ABB RobotStudio station: Solution_20200508-184500.rsstn

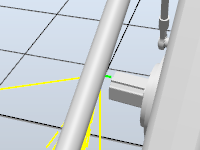
Station Solution (saved by RobotStudio 7.0.8743.626)
Controller Controller
  mechanical unit ROB_1: IRB120_3_58__01, 6 joints, base frame (-200, 0, 800) mm
  mechanical unit ROB_2: IRB120_3_58__01_2, 6 joints, base frame (200, 0, 800) mm, rotated rx 0 ry 0 rz 180 deg
  mechanical unit ROB_3: IRB760_450_318__01, 6 joints, base frame (0, 4000, 0) mm
Layout (positions relative to the parent item):
  - IRB120_3_58__01 [mechanism, from Robots\IRB120_3_58_G_01.rslib] at (-200, 0, 800) mm; joint values [0, -0.7948, 0.351, 0, 2.0145, 0] (rad or m)
  - IRB120_3_58__01_2 [mechanism, from Robots\IRB120_3_58_G_01.rslib] at (200, 0, 800) mm, rotated rx 0 ry 0 rz 180 deg; joint values [0, -0.7948, 0.351, 0, 2.0145, 0] (rad or m)
  - IRB760_450_318__01 [mechanism, from Robots\IRB760_450_318__01.rslib] at (0, 4000, 0) mm; joint values [-0.1057, 0.2404, 0.623, -1.118] (rad or m)
  - Part_1 [part]
  - Tool_1 [mechanism] at (-150, 0, 1400) mm, rotated rx 180 ry 0 rz 180 deg
      TCP Tool1 at (0, 0, 0) mm
      links: SimpleGripper
  - Tool_2 [mechanism] at (150, 0, 1400) mm, rotated rx 180 ry 0 rz 0 deg
      TCP Tool_2 at (0, 0, 0) mm
      links: SimpleGripper
  - Tool_3 [mechanism] at (1980, 3790, 1000) mm, rotated rx 180 ry 0 rz -122 deg
      TCP Tool_3 at (0, 0, 0) mm
      links: SimpleGripper
Attachment: Tool_1 is attached to IRB120_3_58__01 / Link6
Attachment: Tool_2 is attached to IRB120_3_58__01_2 / Link6
Attachment: Tool_3 is attached to IRB760_450_318__01 / Link6
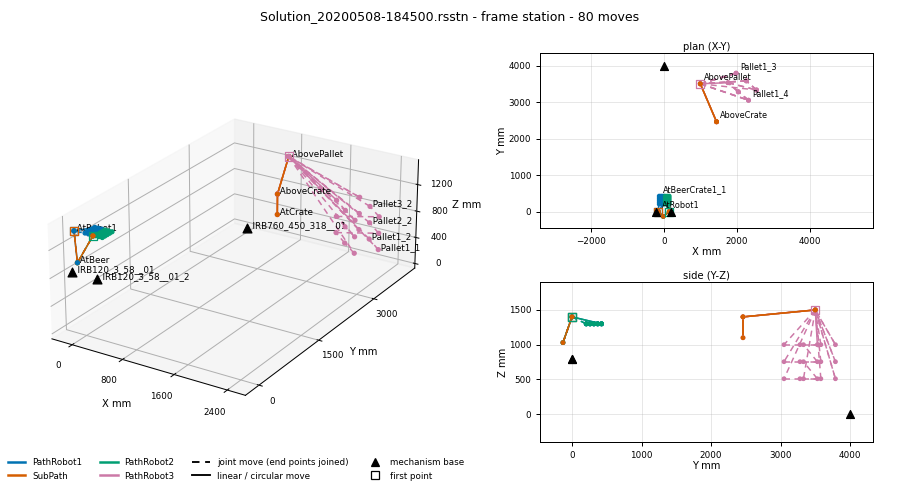
[picture p0: tool path of Solution_20200508-184500.rsstn in frame station, 80 of 80 moves have a stored position in this frame; points joined in program order, loops and branches not executed]
Targets, tools, work objects and paths stored in the station, written as RAPID:
! task T_ROB1
MODULE CalibData
  PERS tooldata Tool1:=[TRUE,[[0,0,0],[1,0,0,0]],[1,[0,0,1],[1,0,0,0],0,0,0]];
ENDMODULE

! task T_ROB1
MODULE Module1
  CONST robtarget AtBeer:=[[-15,-130,1030],[0,0,1,0],[-1,0,-1,0],[9E+09,9E+09,9E+09,9E+09,9E+09,9E+09]];
  CONST robtarget AtRobot1:=[[-150,0,1400],[0,0,1,0],[0,0,0,0],[9E+09,9E+09,9E+09,9E+09,9E+09,9E+09]];
  CONST robtarget AtBeerCrate1_1:=[[-125,425,1300],[0,0,1,0],[0,0,0,0],[9E+09,9E+09,9E+09,9E+09,9E+09,9E+09]];
  CONST robtarget AtBeerCrate1_2:=[[-125,370,1300],[0,0,1,0],[0,0,0,0],[9E+09,9E+09,9E+09,9E+09,9E+09,9E+09]];
  CONST robtarget AtBeerCrate1_3:=[[-125,315,1300],[0,0,1,0],[0,0,0,0],[9E+09,9E+09,9E+09,9E+09,9E+09,9E+09]];
  CONST robtarget AtBeerCrate1_4:=[[-125,260,1300],[0,0,1,0],[0,0,0,0],[9E+09,9E+09,9E+09,9E+09,9E+09,9E+09]];
  CONST robtarget AtBeerCrate1_5:=[[-125,205,1300],[0,0,1,0],[0,0,0,0],[9E+09,9E+09,9E+09,9E+09,9E+09,9E+09]];
  CONST robtarget AtBeerCrate2_1:=[[-70,425,1300],[0,0,1,0],[0,0,0,0],[9E+09,9E+09,9E+09,9E+09,9E+09,9E+09]];
  CONST robtarget AtBeerCrate2_2:=[[-70,370,1300],[0,0,1,0],[0,0,0,0],[9E+09,9E+09,9E+09,9E+09,9E+09,9E+09]];
  CONST robtarget AtBeerCrate2_3:=[[-70,315,1300],[0,0,1,0],[0,0,0,0],[9E+09,9E+09,9E+09,9E+09,9E+09,9E+09]];
  CONST robtarget AtBeerCrate2_4:=[[-70,260,1300],[0,0,1,0],[0,0,0,0],[9E+09,9E+09,9E+09,9E+09,9E+09,9E+09]];
  CONST robtarget AtBeerCrate2_5:=[[-70,205,1300],[0,0,1,0],[0,0,0,0],[9E+09,9E+09,9E+09,9E+09,9E+09,9E+09]];
  CONST robtarget AtBeerCrate3_1:=[[-15,425,1300],[0,0,1,0],[0,0,0,0],[9E+09,9E+09,9E+09,9E+09,9E+09,9E+09]];
  CONST robtarget AtBeerCrate3_2:=[[-15,370,1300],[0,0,1,0],[0,0,0,0],[9E+09,9E+09,9E+09,9E+09,9E+09,9E+09]];
  CONST robtarget AtBeerCrate3_3:=[[-15,315,1300],[0,0,1,0],[0,0,0,0],[9E+09,9E+09,9E+09,9E+09,9E+09,9E+09]];
  CONST robtarget AtBeerCrate3_4:=[[-15,260,1300],[0,0,1,0],[0,0,0,0],[9E+09,9E+09,9E+09,9E+09,9E+09,9E+09]];
  CONST robtarget AtBeerCrate3_5:=[[-15,205,1300],[0,0,1,0],[0,0,0,0],[9E+09,9E+09,9E+09,9E+09,9E+09,9E+09]];
  CONST robtarget Target_10:=[[-149.999964851,0,1400.000061087],[-0.000000052,0,1,0],[0,0,0,0],[9E+09,9E+09,9E+09,9E+09,9E+09,9E+09]];
  PROC main()
    PathRobot1;
  ENDPROC
  PROC PathRobot1()
    SetDO DoCrateComplete,0;
    WaitDI Di1CrateReadyForFilling,1;
    MoveJ AtRobot1,v2000,z100,Tool1\WObj:=wobj0;
    MoveL AtBeer,v2000,fine,Tool1\WObj:=wobj0;
    SetDO Do1Gripper,1;
    WaitTime 0.3;
    MoveJ AtRobot1,v2000,z100,Tool1\WObj:=wobj0;
    MoveL AtBeerCrate1_1,v2000,fine,Tool1\WObj:=wobj0;
    SubPath;
    MoveL AtBeerCrate1_2,v2000,fine,Tool1\WObj:=wobj0;
    SubPath;
    MoveL AtBeerCrate1_3,v2000,fine,Tool1\WObj:=wobj0;
    SubPath;
    MoveL AtBeerCrate1_4,v2000,fine,Tool1\WObj:=wobj0;
    SubPath;
    MoveL AtBeerCrate1_5,v2000,fine,Tool1\WObj:=wobj0;
    SubPath;
    MoveL AtBeerCrate2_1,v2000,fine,Tool1\WObj:=wobj0;
    SubPath;
    MoveL AtBeerCrate2_2,v2000,fine,Tool1\WObj:=wobj0;
    SubPath;
    MoveL AtBeerCrate2_3,v2000,fine,Tool1\WObj:=wobj0;
    SubPath;
    MoveL AtBeerCrate2_4,v2000,fine,Tool1\WObj:=wobj0;
    SubPath;
    MoveL AtBeerCrate2_5,v2000,fine,Tool1\WObj:=wobj0;
    SubPath;
    MoveL AtBeerCrate3_1,v2000,fine,Tool1\WObj:=wobj0;
    SubPath;
    MoveL AtBeerCrate3_2,v2000,fine,Tool1\WObj:=wobj0;
    SubPath;
    MoveL AtBeerCrate3_3,v2000,fine,Tool1\WObj:=wobj0;
    SubPath;
    MoveL AtBeerCrate3_4,v2000,fine,Tool1\WObj:=wobj0;
    SubPath;
    MoveL AtBeerCrate3_5,v2000,fine,Tool1\WObj:=wobj0;
    SetDO Do1Gripper,0;
    WaitTime 0.3;
    MoveJ AtRobot1,v2000,z100,Tool1\WObj:=wobj0;
    SetDO DoCrateComplete,1;
    WaitTime 0.3;
  ENDPROC
  PROC SubPath()
    SetDO Do1Gripper,0;
    WaitTime 0.3;
    MoveJ AtRobot1,v2000,z100,Tool1\WObj:=wobj0;
    MoveL AtBeer,v2000,fine,Tool1\WObj:=wobj0;
    SetDO Do1Gripper,1;
    WaitTime 0.3;
    MoveJ AtRobot1,v2000,z100,Tool1\WObj:=wobj0;
  ENDPROC
ENDMODULE

! task T_ROB2
MODULE Module1
  CONST robtarget AtBeer:=[[-15,-130,1030],[0,1,0,0],[0,0,0,0],[9E+09,9E+09,9E+09,9E+09,9E+09,9E+09]];
  CONST robtarget AtRobot2:=[[150,0,1400],[0,1,0,0],[0,0,0,0],[9E+09,9E+09,9E+09,9E+09,9E+09,9E+09]];
  CONST robtarget AtBeerCrate4_1:=[[40,425,1300],[0,1,0,0],[-1,0,-1,0],[9E+09,9E+09,9E+09,9E+09,9E+09,9E+09]];
  CONST robtarget AtBeerCrate4_2:=[[40,370,1300],[0,1,0,0],[-1,0,-1,0],[9E+09,9E+09,9E+09,9E+09,9E+09,9E+09]];
  CONST robtarget AtBeerCrate4_3:=[[40,315,1300],[0,1,0,0],[-1,0,-1,0],[9E+09,9E+09,9E+09,9E+09,9E+09,9E+09]];
  CONST robtarget AtBeerCrate4_4:=[[40,260,1300],[0,1,0,0],[-1,0,-1,0],[9E+09,9E+09,9E+09,9E+09,9E+09,9E+09]];
  CONST robtarget AtBeerCrate4_5:=[[40,205,1300],[0,1,0,0],[-1,0,-1,0],[9E+09,9E+09,9E+09,9E+09,9E+09,9E+09]];
  CONST robtarget AtBeerCrate5_1:=[[95,425,1300],[0,1,0,0],[-1,0,-1,0],[9E+09,9E+09,9E+09,9E+09,9E+09,9E+09]];
  CONST robtarget AtBeerCrate5_2:=[[95,370,1300],[0,1,0,0],[-1,0,-1,0],[9E+09,9E+09,9E+09,9E+09,9E+09,9E+09]];
  CONST robtarget AtBeerCrate5_3:=[[95,315,1300],[0,1,0,0],[-1,0,-1,0],[9E+09,9E+09,9E+09,9E+09,9E+09,9E+09]];
  CONST robtarget AtBeerCrate5_4:=[[95,260,1300],[0,1,0,0],[-1,0,-1,0],[9E+09,9E+09,9E+09,9E+09,9E+09,9E+09]];
  CONST robtarget AtBeerCrate5_5:=[[95,205,1300],[0,1,0,0],[0,0,0,0],[9E+09,9E+09,9E+09,9E+09,9E+09,9E+09]];
  CONST robtarget AtBeerCrate6_1:=[[150,425,1300],[0,1,0,0],[0,0,0,0],[9E+09,9E+09,9E+09,9E+09,9E+09,9E+09]];
  CONST robtarget AtBeerCrate6_2:=[[150,370,1300],[0,1,0,0],[0,0,0,0],[9E+09,9E+09,9E+09,9E+09,9E+09,9E+09]];
  CONST robtarget AtBeerCrate6_3:=[[150,315,1300],[0,1,0,0],[0,0,0,0],[9E+09,9E+09,9E+09,9E+09,9E+09,9E+09]];
  CONST robtarget AtBeerCrate6_4:=[[150,260,1300],[0,1,0,0],[0,0,0,0],[9E+09,9E+09,9E+09,9E+09,9E+09,9E+09]];
  CONST robtarget AtBeerCrate6_5:=[[150,205,1300],[0,1,0,0],[0,0,0,0],[9E+09,9E+09,9E+09,9E+09,9E+09,9E+09]];
  PROC main()
    PathRobot2;
  ENDPROC
  PROC PathRobot2()
    WaitDI Di1CrateReadyForFilling,1;
    MoveJ AtRobot2,v2000,z100,Tool2\WObj:=wobj0;
    WaitTime 1.5;
    MoveL AtBeer,v2000,fine,Tool2\WObj:=wobj0;
    SetDO Do2Gripper,0;
    WaitTime 0.3;
    MoveJ AtRobot2,v2000,z100,Tool2\WObj:=wobj0;
    MoveL AtBeerCrate4_1,v2000,fine,Tool2\WObj:=wobj0;
    SubPath;
    MoveL AtBeerCrate4_2,v2000,fine,Tool2\WObj:=wobj0;
    SubPath;
    MoveL AtBeerCrate4_3,v2000,fine,Tool2\WObj:=wobj0;
    SubPath;
    MoveL AtBeerCrate4_4,v2000,fine,Tool2\WObj:=wobj0;
    SubPath;
    MoveL AtBeerCrate4_5,v2000,fine,Tool2\WObj:=wobj0;
    SubPath;
    MoveL AtBeerCrate5_1,v2000,fine,Tool2\WObj:=wobj0;
    SubPath;
    MoveL AtBeerCrate5_2,v2000,fine,Tool2\WObj:=wobj0;
    SubPath;
    MoveL AtBeerCrate5_3,v2000,fine,Tool2\WObj:=wobj0;
    SubPath;
    MoveL AtBeerCrate5_4,v2000,fine,Tool2\WObj:=wobj0;
    SubPath;
    MoveL AtBeerCrate5_5,v2000,fine,Tool2\WObj:=wobj0;
    SubPath;
    MoveL AtBeerCrate6_1,v2000,fine,Tool2\WObj:=wobj0;
    SubPath;
    MoveL AtBeerCrate6_2,v2000,fine,Tool2\WObj:=wobj0;
    SubPath;
    MoveL AtBeerCrate6_3,v2000,fine,Tool2\WObj:=wobj0;
    SubPath;
    MoveL AtBeerCrate6_4,v2000,fine,Tool2\WObj:=wobj0;
    SubPath;
    MoveL AtBeerCrate6_5,v2000,fine,Tool2\WObj:=wobj0;
    SetDO Do2Gripper,0;
    WaitTime 0.3;
    MoveJ AtRobot2,v2000,z100,Tool2\WObj:=wobj0;
  ENDPROC
  PROC SubPath()
    SetDO Do2Gripper,0;
    WaitTime 0.3;
    MoveJ AtRobot2,v2000,z100,Tool2\WObj:=wobj0;
    MoveL AtBeer,v2000,fine,Tool2\WObj:=wobj0;
    SetDO Do2Gripper,1;
    WaitTime 0.3;
    MoveJ AtRobot2,v2000,z100,Tool2\WObj:=wobj0;
  ENDPROC
ENDMODULE

! task T_ROB2
MODULE CalibData
  PERS tooldata Tool2:=[TRUE,[[0,0,0],[1,0,0,0]],[1,[0,0,1],[1,0,0,0],0,0,0]];
  PERS tooldata Tool_2:=[TRUE,[[0,0,0],[1,0,0,0]],[1,[0,0,1],[1,0,0,0],0,0,0]];
ENDMODULE

! task T_ROB3
MODULE CalibData
  PERS tooldata Tool_3:=[TRUE,[[0,0,0],[1,0,0,0]],[1,[0,0,1],[1,0,0,0],0,0,0]];
ENDMODULE

! task T_ROB3
MODULE Module1
  CONST robtarget AtCrate:=[[1445,2460,1100],[0,0,1,0],[0,0,0,0],[9E+09,9E+09,9E+09,9E+09,9E+09,9E+09]];
  CONST robtarget AbovePallet:=[[1000,3500,1500],[0,0,1,0],[0,0,0,0],[9E+09,9E+09,9E+09,9E+09,9E+09,9E+09]];
  CONST robtarget Pallet1_6:=[[1760,3530,510],[0,0.275637356,0.961261696,0],[0,0,0,0],[9E+09,9E+09,9E+09,9E+09,9E+09,9E+09]];
  CONST robtarget Pallet1_5:=[[2040,3280,510],[0,0.275637356,0.961261696,0],[0,0,0,0],[9E+09,9E+09,9E+09,9E+09,9E+09,9E+09]];
  CONST robtarget Pallet1_4:=[[2320,3050,510],[0,-0.48480962,0.874619707,0],[0,0,0,0],[9E+09,9E+09,9E+09,9E+09,9E+09,9E+09]];
  CONST robtarget Pallet1_1:=[[2540,3330,510],[0,0.275637356,0.961261696,0],[0,0,0,0],[9E+09,9E+09,9E+09,9E+09,9E+09,9E+09]];
  CONST robtarget Pallet1_2:=[[2260,3580,510],[0,0.275637356,0.961261696,0],[0,0,0,0],[9E+09,9E+09,9E+09,9E+09,9E+09,9E+09]];
  CONST robtarget Pallet1_3:=[[1980,3790,510],[0,-0.48480962,0.874619707,0],[0,0,0,0],[9E+09,9E+09,9E+09,9E+09,9E+09,9E+09]];
  CONST robtarget AboveCrate:=[[1445,2460,1400],[0,0,1,0],[0,0,0,0],[9E+09,9E+09,9E+09,9E+09,9E+09,9E+09]];
  CONST robtarget Pallet2_1:=[[2540,3330,755],[0,0.275637356,0.961261696,0],[0,0,0,0],[9E+09,9E+09,9E+09,9E+09,9E+09,9E+09]];
  CONST robtarget Pallet2_2:=[[2260,3580,755],[0,0.275637356,0.961261696,0],[0,0,0,0],[9E+09,9E+09,9E+09,9E+09,9E+09,9E+09]];
  CONST robtarget Pallet2_3:=[[1980,3790,755],[0,-0.48480962,0.874619707,0],[0,0,0,0],[9E+09,9E+09,9E+09,9E+09,9E+09,9E+09]];
  CONST robtarget Pallet2_4:=[[2320,3050,755],[0,-0.48480962,0.874619707,0],[0,0,0,0],[9E+09,9E+09,9E+09,9E+09,9E+09,9E+09]];
  CONST robtarget Pallet2_5:=[[2040,3280,755],[0,0.275637356,0.961261696,0],[0,0,0,0],[9E+09,9E+09,9E+09,9E+09,9E+09,9E+09]];
  CONST robtarget Pallet2_6:=[[1760,3530,755],[0,0.275637356,0.961261696,0],[0,0,0,0],[9E+09,9E+09,9E+09,9E+09,9E+09,9E+09]];
  CONST robtarget Pallet3_1:=[[2540,3330,1000],[0,0.275637356,0.961261696,0],[0,0,0,0],[9E+09,9E+09,9E+09,9E+09,9E+09,9E+09]];
  CONST robtarget Pallet3_2:=[[2260,3580,1000],[0,0.275637356,0.961261696,0],[0,0,0,0],[9E+09,9E+09,9E+09,9E+09,9E+09,9E+09]];
  CONST robtarget Pallet3_3:=[[1980,3790,1000],[0,-0.48480962,0.874619707,0],[0,0,0,0],[9E+09,9E+09,9E+09,9E+09,9E+09,9E+09]];
  CONST robtarget Pallet3_4:=[[2320,3050,1000],[0,-0.48480962,0.874619707,0],[0,0,0,0],[9E+09,9E+09,9E+09,9E+09,9E+09,9E+09]];
  CONST robtarget Pallet3_5:=[[2040,3280,1000],[0,0.275637356,0.961261696,0],[0,0,0,0],[9E+09,9E+09,9E+09,9E+09,9E+09,9E+09]];
  CONST robtarget Pallet3_6:=[[1760,3530,1000],[0,0.275637356,0.961261696,0],[0,0,0,0],[9E+09,9E+09,9E+09,9E+09,9E+09,9E+09]];
  CONST robtarget AbovePalletRotated:=[[1000,3500,1500],[0,0,1,0],[0,0,0,0],[9E+09,9E+09,9E+09,9E+09,9E+09,9E+09]];
  PROC PathRobot3()
    SetDO DoPalletComplete,0;
    MoveJ AbovePallet,v2000,z100,Tool_3\WObj:=wobj0;
    MoveL AboveCrate,v2000,z100,Tool_3\WObj:=wobj0;
    WaitDI Di2CrateReadyForPacking,1;
    MoveL AtCrate,v2000,fine,Tool_3\WObj:=wobj0;
    SetDO Do3Gripper,1;
    WaitTime 0.3;
    MoveL AboveCrate,v2000,z100,Tool_3\WObj:=wobj0;
    MoveL AbovePallet,v2000,z100,Tool_3\WObj:=wobj0;
    MoveJ Pallet1_1,v2000,fine,Tool_3\WObj:=wobj0;
    SubPath;
    MoveJ Pallet1_2,v2000,fine,Tool_3\WObj:=wobj0;
    SubPath;
    MoveJ AbovePalletRotated,v2000,z100,Tool_3\WObj:=wobj0;
    MoveJ Pallet1_3,v2000,fine,Tool_3\WObj:=wobj0;
    SubPath;
    MoveJ AbovePalletRotated,v2000,z100,Tool_3\WObj:=wobj0;
    MoveJ Pallet1_4,v2000,fine,Tool_3\WObj:=wobj0;
    SubPath;
    MoveJ Pallet1_5,v2000,fine,Tool_3\WObj:=wobj0;
    SubPath;
    MoveJ Pallet1_6,v2000,fine,Tool_3\WObj:=wobj0;
    SubPath;
    MoveJ Pallet2_1,v2000,fine,Tool_3\WObj:=wobj0;
    SubPath;
    MoveJ Pallet2_2,v2000,fine,Tool_3\WObj:=wobj0;
    SubPath;
    MoveJ AbovePalletRotated,v2000,z100,Tool_3\WObj:=wobj0;
    MoveJ Pallet2_3,v2000,fine,Tool_3\WObj:=wobj0;
    SubPath;
    MoveJ AbovePalletRotated,v2000,z100,Tool_3\WObj:=wobj0;
    MoveJ Pallet2_4,v2000,fine,Tool_3\WObj:=wobj0;
    SubPath;
    MoveJ Pallet2_5,v2000,fine,Tool_3\WObj:=wobj0;
    SubPath;
    MoveJ Pallet2_6,v2000,fine,Tool_3\WObj:=wobj0;
    SubPath;
    MoveJ Pallet3_1,v2000,fine,Tool_3\WObj:=wobj0;
    SubPath;
    MoveJ Pallet3_2,v2000,fine,Tool_3\WObj:=wobj0;
    SubPath;
    MoveJ AbovePalletRotated,v2000,z100,Tool_3\WObj:=wobj0;
    MoveJ Pallet3_3,v2000,fine,Tool_3\WObj:=wobj0;
    SubPath;
    MoveJ AbovePalletRotated,v2000,z100,Tool_3\WObj:=wobj0;
    MoveJ Pallet3_4,v2000,fine,Tool_3\WObj:=wobj0;
    SubPath;
    MoveJ Pallet3_5,v2000,fine,Tool_3\WObj:=wobj0;
    SubPath;
    MoveJ Pallet3_6,v2000,fine,Tool_3\WObj:=wobj0;
    SetDO Do3Gripper,0;
    WaitTime 0.3;
    MoveL AbovePallet,v2000,z100,Tool_3\WObj:=wobj0;
    MoveJ AboveCrate,v2000,z100,Tool_3\WObj:=wobj0;
    SetDO DoPalletComplete,1;
  ENDPROC
  PROC SubPath()
    SetDO Do3Gripper,0;
    WaitTime 0.3;
    MoveJ AbovePallet,v2000,z100,Tool_3\WObj:=wobj0;
    MoveL AboveCrate,v2000,z100,Tool_3\WObj:=wobj0;
    WaitDI Di2CrateReadyForPacking,1;
    MoveL AtCrate,v2000,fine,Tool_3\WObj:=wobj0;
    SetDO Do3Gripper,1;
    WaitTime 0.3;
    MoveL AboveCrate,v2000,z100,Tool_3\WObj:=wobj0;
    MoveL AbovePallet,v2000,z100,Tool_3\WObj:=wobj0;
  ENDPROC
  PROC main()
    PathRobot3;
  ENDPROC
ENDMODULE

